PROGRAM MAIN
VAR
END_VAR

END_PROGRAM

(* stored: Version 1.1.0.1
   POU MAIN: Id {5f753085-44ac-4e13-8c70-ae76b4eaba58} *)
